TEXTLIST E_MessageNumbers
  0 = 'NA_NoMessage'
  1 = 'FF_Unknown'
  2 = 'FF_NoCommunication'
  3 = 'FF_ComunicationFault'
  4 = 'FF_Overload'
  5 = 'FF_EncoderFault'
  6 = 'FF_SlaveFault'
  7 = 'FF_AxisFault'
  8 = 'FF_DriveFault'
  9 = 'FF_Collision'
  100 = 'CF_FeedbackFault'
  101 = 'CF_WrongDirection'
  102 = 'CF_MoveToFast'
  103 = 'CF_MoveToSlow'
  104 = 'CF_WrongPosition'
  105 = 'CF_Obstruction'
  200 = 'MC_WaitingForproduct'
  201 = 'MC_WaitingForOperator'
  202 = 'MC_WaitingForModule'
  203 = 'MC_WaitingForMaster'
  204 = 'MC_WaitingForSlave'
  205 = 'MC_WrongPosition'
  300 = 'OM_AlmostEmpty'
  301 = 'OM_Finished'
  302 = 'OM_ready'
  900 = 'FF_MessageTest'
  901 = 'CF_MessageTest'
  902 = 'MC_MessageTest'
  903 = 'OM_MessageTest'
   = ''
END_TEXTLIST

(* stored: Version 1.1.0.1, ProductVersion 3.1.4024.3
   TextList E_MessageNumbers: Id {ea16fe31-2713-4200-b8f9-70b56e66bb6b} *)
